// TIA Portal V20 export
DATA_BLOCK "TESTSEQ"   // DB73
// stored: MemoryReserve 100, Namespace Unit1.Em2
   VAR
      SIM : Bool;
      Job1_ : Array[0..40] of Bool;
      Job2_ : Array[0..40] of Bool;
      Job3_ : Array[0..40] of Bool;
   END_VAR
BEGIN
END_DATA_BLOCK
